INTERFACE ILogger

METHOD Write : STRING
VAR_INPUT
	sMsg    : STRING;
END_VAR
END_METHOD

END_INTERFACE

(* stored: Version 1.1.0.1, ProductVersion 3.1.0.24
   Itf ILogger: Id {14749118-71ce-4f16-889e-971120f50765}
   Method Write: Id {9291435e-f081-4fb5-93ae-57f08b2b3af2} *)
